Yaskawa INFORM job: X4_NOWY2_SPR.JBI

/JOB
//NAME X4_NOWY2_SPR
//POS
///NPOS 273,273,273,16,0,0
///TOOL 0
///POSTYPE PULSE
///PULSE
C00000=1579,-114561,-88072,141,60969,-160
C00001=1579,-126069,-115869,130,72161,-147
C00002=-67532,-124352,-115339,134,72718,-152
C00003=-81630,-76415,-67707,7081,99866,-75616
C00004=-81630,-76414,-67706,7081,99866,-75616
C00005=-84756,-88459,-71994,6618,96608,-76878
C00006=-84756,-88020,-70779,6612,96092,-76905
C00007=-84756,-88291,-71526,6619,96412,-76888
C00008=-86383,-83236,-69405,6430,97828,-77376
C00009=-86383,-82906,-68386,6422,97374,-77400
C00010=-85654,-85197,-69362,6508,96744,-77183
C00011=-88190,-77633,-68794,6246,100461,-77872
C00012=-91609,-64546,-67425,5952,106567,-78770
C00013=-108338,-72557,-69392,19017,102016,-84323
C00014=-103994,-87799,-70649,19047,94316,-83966
C00015=-101720,-95837,-73131,19200,91317,-83621
C00016=-101720,-95093,-71454,19192,90702,-83718
C00017=-101720,-95403,-72147,19196,90955,-83679
C00018=-102509,-90897,-70406,19144,92318,-83747
C00019=-102509,-90529,-69509,19136,91974,-83801
C00020=-102070,-93055,-70499,19166,91217,-83763
C00021=-103193,-87364,-70534,19135,94271,-83684
C00022=-105000,-74500,-64879,19101,97659,-83800
C00023=-113069,-60767,-53247,26239,106025,-84622
C00024=-112828,-63942,-52646,27281,108527,-83919
C00025=-112433,-69525,-54608,27546,108328,-83811
C00026=-112433,-69174,-53580,27467,107925,-83912
C00027=-112433,-68598,-51946,27347,107292,-84070
C00028=-112433,-68839,-52622,27396,107553,-84005
C00029=-112673,-65386,-50917,27452,108279,-83921
C00030=-112673,-65100,-50066,27387,107943,-84004
C00031=-112560,-66748,-50889,27360,107600,-84043
C00032=-112776,-63836,-50109,27476,108578,-83887
C00033=-126682,-57830,-51235,23795,116313,-87772
C00034=-91609,-64546,-67425,5952,106567,-78770
C00035=-73590,-134956,-134527,8565,110042,-72105
C00036=-73590,-134956,-134527,8565,110042,-72105
C00037=-85079,-90579,-82104,6699,101738,-76716
C00038=-105233,-99145,-78854,31145,91869,-85162
C00039=-90886,-100639,-75930,30232,80497,-82559
C00040=-84197,-95229,-69335,30102,76988,-80863
C00041=-84197,-94656,-68126,30150,76597,-80967
C00042=-84197,-94979,-68806,30123,76817,-80908
C00043=-86405,-88952,-66471,30068,79053,-81183
C00044=-86405,-88608,-65674,30094,78780,-81256
C00045=-85194,-91982,-67001,30129,77549,-81108
C00046=-89786,-90500,-68269,30172,80536,-82119
C00047=-91499,-86657,-71640,30020,84676,-81700
C00048=-78974,-84836,-79700,7511,102662,-74517
C00049=-78974,-83060,-72035,7396,98889,-74746
C00050=-78731,-83061,-70147,7399,97713,-74732
C00051=-78731,-82586,-68642,7386,97035,-74771
C00052=-78693,-82844,-69189,7365,97187,-74749
C00053=-80468,-78121,-67102,7173,98481,-75288
C00054=-80468,-77948,-66494,7167,98198,-75304
C00055=-79573,-80363,-67572,7265,97545,-75033
C00056=-80252,-78819,-67734,7202,98493,-75213
C00057=-80252,-80316,-73749,7282,101403,-75042
C00058=-98731,-93358,-79222,4709,99471,-81580
C00059=-97921,-96065,-76902,4782,96613,-81409
C00060=-97642,-96671,-75645,4808,95516,-81355
C00061=-97642,-96038,-74155,4803,94926,-81379
C00062=-97642,-96278,-74718,4805,95148,-81370
C00063=-99165,-88824,-71799,4613,97264,-81812
C00064=-99165,-88527,-70990,4608,96920,-81825
C00065=-98316,-92764,-72679,4715,95737,-81578
C00066=-99279,-88707,-72907,4606,98011,-81825
C00067=-99279,-90964,-80150,4662,101298,-81702
C00068=-83031,-73882,-65637,-17912,114082,-77307
C00069=-84799,-81323,-60919,-25592,110942,-77323
C00070=-87066,-81955,-59363,-24887,108536,-77734
C00071=-87066,-80978,-57100,-24746,107724,-77553
C00072=-87066,-81307,-57855,-24792,107993,-77613
C00073=-89010,-75270,-55192,-25677,108733,-78552
C00074=-89010,-74947,-54382,-25621,108431,-78482
C00075=-88073,-77930,-55720,-25197,108074,-78029
C00076=-86155,-69275,-53538,-25095,111477,-78039
C00077=-82305,-66217,-52035,-23871,113209,-76862
C00078=-98731,-93358,-79222,4709,99471,-81580
C00079=-87850,-130184,-128808,6122,98008,-77863
C00080=-131124,-97291,-82060,5244,66687,-6018
C00081=-125790,2337,-22266,13440,105024,83634
C00082=-119533,36956,22492,13071,94512,84678
C00083=-111606,23469,-6781,11265,89839,86812
C00084=-109349,27190,646,10801,86931,87307
C00085=-108816,27234,2830,10703,85564,87368
C00086=-108816,27153,4539,10716,84489,87276
C00087=-108816,27166,4149,10713,84731,87297
C00088=-107956,27551,4528,10540,84587,87578
C00089=-108965,27264,1619,10711,86335,87387
C00090=-111260,52324,24435,15027,98353,88139
C00091=-102462,56667,28820,9286,105586,72437
C00092=-101371,54153,30717,9255,103034,72626
C00093=-101300,53253,30624,9243,102627,72619
C00094=-101300,53374,32279,9201,101680,72548
C00095=-101300,53356,32072,9206,101797,72557
C00096=-100857,47625,25743,9281,102687,72780
C00097=-100773,46580,24617,9295,102831,72821
C00098=-101300,53356,32072,9206,101797,72557
C00099=-102175,52590,31226,9140,102021,72268
C00100=-102630,52208,30804,9106,102134,72116
C00101=-102175,52590,31226,9140,102021,72268
C00102=-99428,22928,-9812,4382,95874,-22555
C00103=-101546,17046,-6787,4678,91283,-23411
C00104=-101546,16945,-5416,4675,90390,-23444
C00105=-101514,16566,-4490,4670,89624,-23462
C00106=-101514,16574,-4727,4671,89774,-23457
C00107=-101796,19478,-2026,4708,89621,-23556
C00108=-101749,19095,-4432,4706,90897,-23492
C00109=-101749,19375,-7041,4715,92641,-23427
C00110=-101749,19375,-7041,4715,92641,-23427
C00111=-102981,33005,7118,6834,98538,-23358
C00112=-102660,29046,5283,6805,97611,-23301
C00113=-102660,29002,6609,6789,96777,-23347
C00114=-102660,29022,5897,6798,97224,-23322
C00115=-102541,27735,4980,6792,97060,-7882
C00116=-102724,29871,7085,6794,96879,-7954
C00117=-102669,29379,3677,6831,98706,-7835
C00118=-102669,30744,-3500,6979,103789,-7548
C00119=-89085,-61640,-68335,6227,95184,-3424
C00120=-129723,10180,-8133,7222,98462,-17027
C00121=-105913,33806,-16630,-33387,116609,-16888
C00122=-114766,23108,-3420,-30164,101829,-15972
C00123=-126000,19507,-6631,-29272,96237,-18805
C00124=-125928,21918,3078,-29245,93808,-18174
C00125=-125928,21960,4203,-29214,93219,-18024
C00126=-125927,21943,3808,-29209,93425,-18075
C00127=-125864,24512,6268,-29206,93280,-18014
C00128=-125884,23639,4506,-29235,93832,-18161
C00129=-125884,23787,-988,-29454,96866,-18937
C00130=-117200,23539,-1226,-29926,99884,-16393
C00131=-117161,21121,72,-29726,98116,-15912
C00132=-117144,20144,1246,-29621,97051,-15628
C00133=-117144,20183,2462,-29564,96414,-15463
C00134=-117144,20179,2362,-29568,96466,-15476
C00135=-117212,24135,6125,-29546,96194,-15431
C00136=-117202,23528,1396,-29761,98470,-16021
C00137=-113126,35471,9950,-29950,100652,-15017
C00138=-113126,35383,12410,-29782,99292,-14657
C00139=-113602,35282,14657,-29641,97872,-14469
C00140=-113602,35350,16056,-29571,97148,-14281
C00141=-113602,35312,15354,-29605,97509,-14375
C00142=-114294,35130,15170,-29602,97286,-14585
C00143=-113391,35371,15415,-29607,97577,-14310
C00144=-113626,42883,17073,-29878,99977,-15031
C00145=-136877,41374,10058,10283,103905,-75706
C00146=-141001,35831,8537,10150,102526,-77247
C00147=-140132,39057,14516,9459,103035,-76976
C00148=-140132,39037,16298,9412,101942,-77061
C00149=-140132,39036,16078,9417,102075,-77051
C00150=-140481,35058,11996,9419,102579,-77132
C00151=-140132,39036,16078,9417,102075,-77051
C00152=-138905,38111,15122,9481,102046,-76624
C00153=-140132,39045,14975,9447,102749,-76998
C00154=-140132,39114,13214,9498,103853,-76912
C00155=-141320,33353,7524,13959,97601,-77374
C00156=-139853,30861,8005,10213,95427,-68773
C00157=-139850,30231,7379,10216,95489,-68766
C00158=-141726,26843,4526,13791,96694,-77632
C00159=-141207,31872,9522,12754,100191,-77170
C00160=-131838,40307,17400,-3069,104254,-75449
C00161=-120717,39791,20254,-22002,103322,-74072
C00162=-123241,41817,22993,-23858,102713,-75145
C00163=-120965,41759,25023,-29185,101758,-74907
C00164=-121023,25271,5223,-28433,95326,-73297
C00165=-120372,33506,8504,-28624,97501,-73589
C00166=-120372,33506,8504,-28624,97501,-7388
C00167=-114011,28987,3831,-29482,105348,-6966
C00168=-127301,22883,-362,-9290,98378,-8800
C00169=-130383,22892,110,-12210,96784,-9925
C00170=-119117,21486,5591,-32037,93907,-6966
C00171=-117872,21036,1539,-32238,96305,-7157
C00172=-135561,25772,-1454,-7801,99682,-11540
C00173=-135461,26025,2407,-7746,97466,-11367
C00174=-129197,23357,2778,-20865,94605,-10044
C00175=-129563,23522,5318,-26932,92135,-10188
C00176=-126533,22338,1333,-27220,94758,-9659
C00177=-115633,44815,18495,-18996,108364,22675
C00178=-114062,50158,32326,-24769,103985,23625
C00179=-114261,61004,44440,-24574,102207,23931
C00180=-113327,59043,39697,-24681,104230,23854
C00181=-113549,43239,22387,-25049,106471,23276
C00182=-113959,36250,17368,-26116,100180,17331
C00183=-113750,32141,13338,-26671,97959,14884
C00184=-113784,32033,10394,-26825,99526,14508
C00185=-112924,58292,37776,-24734,105077,23825
C00186=-109456,25709,2980,-23794,97137,26657
C00187=-118237,30699,-4511,6400,110959,24971
C00188=-106534,-87247,-110627,560,89262,27492
C00189=-106534,-87247,-110627,560,89262,27492
C00190=-103790,-60662,-71601,3492,92371,24893
C00191=-90072,-46297,-51679,19403,82444,29914
C00192=-89225,-25796,-38496,19051,95364,28629
C00193=-82968,-19569,-33829,18693,94249,30668
C00194=-92316,-28208,-34631,31848,87681,26801
C00195=-93212,-29211,-40642,31971,90742,27310
C00196=-74629,-7827,-31935,11254,101997,33705
C00197=-71338,-2997,-23236,6798,101883,34323
C00198=-78936,-14568,-30649,16904,94877,32031
C00199=-82428,-18766,-28557,29607,85533,29992
C00200=-85091,-23046,-35219,29948,88128,29642
C00201=-83302,-13788,-26964,29706,87219,30090
C00202=-84406,-14503,-30600,29861,89239,30192
C00203=-85356,-5858,-28119,20956,91780,-33865
C00204=-81588,1907,-17110,16920,91332,-34481
C00205=-80085,-4136,-22119,16745,91007,-34003
C00206=-79500,-6857,-23987,16670,90650,-33848
C00207=-76840,-15565,-30031,18766,92661,-32418
C00208=-81974,-12051,-30981,19262,96095,-33689
C00209=-98247,-31422,-44950,19682,96659,-36405
C00210=-99612,-12458,-27594,19698,96098,-36983
C00211=-98475,-20893,-33899,19626,95400,-36692
C00212=-97436,-32531,-42916,18662,91677,-32211
C00213=-95696,-34091,-42802,18103,89563,-30497
C00214=-96230,-30895,-40673,18159,89998,-30622
C00215=-92776,-41331,-47434,14269,83214,-21666
C00216=-93749,-43799,-52657,14401,85273,-21763
C00217=-91043,-39779,-53377,13904,87247,-20611
C00218=-86158,-7385,-30463,15366,102993,-69398
C00219=-78323,6041,-20316,6463,111515,-89101
C00220=-75958,-7074,-26718,1279,101463,-89171
C00221=-73720,-14383,-32408,1291,101175,-88413
C00222=-73707,-14423,-32438,1291,101173,-88409
C00223=-74501,-16417,-33720,1350,100398,-77182
C00224=-81364,-12014,-29075,8477,103574,-60369
C00225=-76974,-6126,-24441,8683,103288,-58863
C00226=-85840,-5383,-30241,8443,108111,-61612
C00227=-85618,-23129,-54211,-23,98050,-63088
C00228=-77730,-75302,-67065,7588,99691,-74263
C00229=-69151,-69068,-61329,2748,102842,-72431
C00230=-87447,-85862,-67970,-5918,101111,-78781
C00231=-86539,-83533,-63306,-15976,104237,-78477
C00232=-79657,-74315,-62077,-14413,109372,-76594
C00233=-66263,-128090,-130023,-6185,104579,-72041
C00234=-66263,-128090,-130023,-6185,104579,-72041
C00235=-94568,-90015,-76427,-6942,102962,-81955
C00236=-117602,-94880,-71794,-18297,96358,-89322
C00237=-121559,-93963,-69420,-18891,94518,-90455
C00238=-120999,-73428,-51402,-33795,103006,-79102
C00239=-123309,-67068,-41693,-44286,101999,-75160
C00240=-127601,-64996,-39493,-46701,100367,-75399
C00241=-114717,-64735,-41398,-43474,107786,-72608
C00242=-113328,-78138,-63059,-20614,107376,-72751
C00243=-119967,-79989,-67356,5538,106972,-75179
C00244=-119600,-81312,-64641,5556,104608,-75155
C00245=-101370,-77587,-62989,10017,103725,-68716
C00246=-107781,-79603,-61547,20378,100372,-71634
C00247=-114949,-81063,-65452,19014,103658,-73736
C00248=-107597,-133050,-132520,1199,109480,-70827
C00249=-107600,-133050,-132519,1199,109480,-70827
C00250=-111097,-94755,-74427,15472,95771,-72593
C00251=-108511,-92825,-70401,15771,93843,-71925
C00252=-108472,-92930,-69979,15769,93534,-71951
C00253=-101455,-63185,-52092,14913,110854,-65885
C00254=-99527,-62495,-51665,15536,110582,-65187
C00255=-84477,-52236,-46062,20087,109018,-59662
C00256=-81486,-46306,-41350,23406,108929,-56767
C00257=-85967,-47236,-42901,22323,110616,-58192
C00258=-110623,-74300,-66049,9174,91324,-69507
C00259=-118006,-113386,-124466,9637,107827,-70792
C00260=-118006,-113386,-124466,9637,107827,-70792
C00261=-104411,-100441,-71960,6543,87095,-88178
C00262=-104969,-99438,-67477,6508,84909,-88479
C00263=-110340,-97663,-63190,-18251,87254,-88347
C00264=-100177,-101375,-72775,-10447,90542,-85701
C00265=-127322,-146784,-131564,384,102103,-77635
C00266=-127322,-146784,-131564,384,102103,-77635
C00267=-128828,-100845,-70585,1227,88109,-75124
C00268=-127499,-98820,-66694,1376,86733,-74692
C00269=-112766,-97884,-65315,11280,85320,-70490
C00270=-128822,-103835,-77575,9498,91788,-75427
C00271=-146076,-192209,-136001,7129,84184,-81740
C00272=-146076,-192209,-136001,7129,84184,-81740
BC00000=127053,672594,1075229
BC00001=127053,672594,1075229
BC00002=210750,818892,1075229
BC00003=210750,818892,1005167
BC00004=210749,818892,1005164
BC00005=210749,818892,1005161
BC00006=210749,818892,1005161
BC00007=210749,818892,1005161
BC00008=210749,818892,1005161
BC00009=210749,818892,1005161
BC00010=210749,818892,1005161
BC00011=210749,818892,1005161
BC00012=210749,818892,1005161
BC00013=255741,818892,1005161
BC00014=255741,818892,1005161
BC00015=255741,818892,1005161
BC00016=255741,818892,1005161
BC00017=255741,818892,1005161
BC00018=255741,818892,1005161
BC00019=255741,818892,1005161
BC00020=255741,818892,1005161
BC00021=255741,818892,1005161
BC00022=255741,818892,1005161
BC00023=287623,818892,1005161
BC00024=287623,818892,1005161
BC00025=287623,818892,1005161
BC00026=287623,818892,1005161
BC00027=287623,818892,1005161
BC00028=287623,818892,1005161
BC00029=287623,818892,1005161
BC00030=287623,818892,1005161
BC00031=287623,818892,1005161
BC00032=287623,818892,1005161
BC00033=287623,818892,1005161
BC00034=210749,818892,1005161
BC00035=210749,818892,1005161
BC00036=119260,818892,1005161
BC00037=119260,818892,1005161
BC00038=119260,818892,1005161
BC00039=119260,818892,1005161
BC00040=119260,818892,1005161
BC00041=119260,818892,1005161
BC00042=119260,818892,1005161
BC00043=119260,818892,1005161
BC00044=119260,818892,1005161
BC00045=119260,818892,1005161
BC00046=119260,818892,1005161
BC00047=119260,818892,1005161
BC00048=119260,818892,1005157
BC00049=119260,818892,1005157
BC00050=119260,818892,1005157
BC00051=119260,818892,1005157
BC00052=119260,818892,1005157
BC00053=119260,818892,1005157
BC00054=119260,818892,1005157
BC00055=119260,818892,1005157
BC00056=119260,818892,1005157
BC00057=119260,818892,1005157
BC00058=119260,818892,1005157
BC00059=119260,818892,1005157
BC00060=119260,818892,1005157
BC00061=119260,818892,1005157
BC00062=119260,818892,1005157
BC00063=119260,818892,1005157
BC00064=119260,818892,1005157
BC00065=119260,818892,1005157
BC00066=119260,818892,1005157
BC00067=119260,818892,1005157
BC00068=119260,818892,1005157
BC00069=119260,818892,1005157
BC00070=119260,818892,1005157
BC00071=119260,818892,1005157
BC00072=119260,818892,1005157
BC00073=119260,818892,1005157
BC00074=119260,818892,1005157
BC00075=119260,818892,1005157
BC00076=119260,818892,1005157
BC00077=119260,818892,1005157
BC00078=119260,818892,1005157
BC00079=119260,818892,1005157
BC00080=271066,672595,967916
BC00081=271066,672595,967916
BC00082=271066,672595,967916
BC00083=271066,672595,742596
BC00084=271066,672596,742593
BC00085=271066,672596,742593
BC00086=271065,672596,742589
BC00087=271065,672596,742589
BC00088=271065,672596,742589
BC00089=271065,672597,742586
BC00090=271065,672597,742586
BC00091=271065,673087,742586
BC00092=271065,673087,742586
BC00093=271065,673087,742586
BC00094=271065,673087,742586
BC00095=271065,673087,742586
BC00096=271065,673087,742586
BC00097=271065,673087,742586
BC00098=271065,673087,742586
BC00099=271065,673087,742586
BC00100=271065,673087,742586
BC00101=271065,673087,742586
BC00102=271065,673085,742583
BC00103=271065,673085,742583
BC00104=271065,673085,742583
BC00105=271065,673085,742583
BC00106=271065,673085,742583
BC00107=271065,673085,742583
BC00108=271065,673085,742583
BC00109=271065,673085,742583
BC00110=291623,673085,742583
BC00111=291623,673085,742583
BC00112=291623,673085,742583
BC00113=291623,673085,742583
BC00114=291623,673085,742583
BC00115=291623,673085,742583
BC00116=291623,673085,742583
BC00117=291623,673085,742583
BC00118=291623,673085,1054355
BC00119=130801,673085,1059449
BC00120=130802,673083,1031676
BC00121=130802,673083,742569
BC00122=130802,673083,742569
BC00123=130802,673083,742569
BC00124=130802,673083,742569
BC00125=130802,673083,742569
BC00126=130802,673083,742566
BC00127=130802,673083,742566
BC00128=130802,673083,742566
BC00129=130802,673083,742566
BC00130=130802,673083,742566
BC00131=130802,673083,742566
BC00132=130802,673083,742566
BC00133=130802,673083,742566
BC00134=130802,673083,742566
BC00135=130802,673083,742566
BC00136=130802,673083,742566
BC00137=130802,673083,742566
BC00138=130802,673083,742566
BC00139=130802,673083,742566
BC00140=130802,673083,742566
BC00141=130802,673083,742566
BC00142=130802,673083,742566
BC00143=130802,673083,742566
BC00144=130802,673083,742566
BC00145=130802,673083,742566
BC00146=130802,673083,742566
BC00147=130802,673083,742566
BC00148=130802,673083,742566
BC00149=130802,673083,742566
BC00150=130802,673083,742566
BC00151=130802,673083,742566
BC00152=130802,673083,742566
BC00153=130802,673083,742566
BC00154=130802,673083,742566
BC00155=130802,673083,742566
BC00156=130802,673083,742566
BC00157=130802,673083,742566
BC00158=130802,673083,742566
BC00159=130802,673083,742566
BC00160=130802,673083,742566
BC00161=130802,673083,742566
BC00162=130802,673083,742566
BC00163=130802,673083,742566
BC00164=130802,673083,742566
BC00165=130802,673083,742566
BC00166=130802,673083,742566
BC00167=130802,673083,742566
BC00168=130802,673083,742566
BC00169=130802,673083,742566
BC00170=130802,673083,742566
BC00171=130802,673083,742566
BC00172=130802,673083,742566
BC00173=130802,673083,742566
BC00174=130802,673083,742566
BC00175=130802,673083,742566
BC00176=130802,673083,742566
BC00177=130802,673083,742566
BC00178=130802,673083,742566
BC00179=130802,673083,742566
BC00180=130802,673083,742566
BC00181=130802,673083,742566
BC00182=130802,673083,742566
BC00183=130802,673083,742566
BC00184=130802,673083,742566
BC00185=130802,673083,742566
BC00186=130802,673083,742566
BC00187=130802,673083,742566
BC00188=130802,673083,742566
BC00189=239197,673083,742566
BC00190=239197,748715,742566
BC00191=239197,748715,742566
BC00192=239196,748714,742562
BC00193=239196,748714,742562
BC00194=239196,748714,742562
BC00195=239196,748714,742562
BC00196=239196,748714,742562
BC00197=239196,748714,742562
BC00198=239196,748714,742562
BC00199=239196,748714,742562
BC00200=239196,748714,742562
BC00201=239196,748714,742562
BC00202=239196,748714,742559
BC00203=239196,748714,742559
BC00204=239196,748714,742559
BC00205=239196,748714,742559
BC00206=239196,748714,742559
BC00207=239196,748714,742559
BC00208=239196,748714,742559
BC00209=239196,748714,742559
BC00210=239196,748714,742559
BC00211=239196,748714,742559
BC00212=239196,748714,742559
BC00213=239196,748714,742559
BC00214=239196,748714,742559
BC00215=239196,748714,742559
BC00216=239196,748714,742559
BC00217=239196,748714,742559
BC00218=239196,748714,742559
BC00219=239196,748714,742559
BC00220=239196,748714,742559
BC00221=239196,748714,742559
BC00222=239196,748714,742559
BC00223=239196,748714,742559
BC00224=239196,748714,742559
BC00225=239196,748714,742559
BC00226=239196,748714,742559
BC00227=239196,748714,742556
BC00228=210749,818892,1005161
BC00229=210749,818892,1005161
BC00230=210750,818891,1005159
BC00231=210750,818891,1005159
BC00232=210750,818891,1005159
BC00233=210750,818891,1005157
BC00234=123072,818891,1005157
BC00235=123072,818891,1005157
BC00236=162220,818891,1005157
BC00237=162220,818891,1005152
BC00238=162220,818891,1005153
BC00239=162220,818891,1005153
BC00240=162220,818891,1005153
BC00241=162220,818891,1005153
BC00242=162220,818891,1005153
BC00243=162220,818891,1005153
BC00244=162220,818891,1005153
BC00245=162220,818891,1005153
BC00246=162220,818891,1005153
BC00247=162220,818891,1005153
BC00248=162220,818891,1005153
BC00249=264269,818892,1005150
BC00250=264269,818892,1005150
BC00251=264269,818892,1005150
BC00252=264269,818892,1005148
BC00253=264269,818892,1005148
BC00254=264269,818892,1005148
BC00255=264269,818892,1005148
BC00256=264269,818892,1005148
BC00257=264269,818892,1005148
BC00258=264269,818892,1005148
BC00259=264269,818892,1005148
BC00260=150431,818892,1056877
BC00261=150431,818892,1056877
BC00262=150431,818892,1056877
BC00263=150431,818892,1056877
BC00264=150431,818892,1056877
BC00265=150431,818892,1056877
BC00266=276083,818892,1056877
BC00267=276083,818892,1056877
BC00268=276083,818892,1056877
BC00269=276083,818892,1056877
BC00270=276083,818892,1056877
BC00271=276083,818892,1056877
BC00272=276083,684480,1056877
EC00000=-1527674,557300
EC00001=-1527674,557300
EC00002=-1527674,557300
EC00003=-1527674,557300
EC00004=-1527674,557300
EC00005=-1527674,557301
EC00006=-1527674,557301
EC00007=-1527674,557301
EC00008=-1527674,557301
EC00009=-1527674,557301
EC00010=-1527674,557301
EC00011=-1527674,557301
EC00012=-1527674,557301
EC00013=-1527674,557301
EC00014=-1527674,557301
EC00015=-1527674,557301
EC00016=-1527674,557301
EC00017=-1527674,557301
EC00018=-1527674,557301
EC00019=-1527674,557301
EC00020=-1527674,557301
EC00021=-1527674,557301
EC00022=-1527674,557301
EC00023=-1527674,557301
EC00024=-1527674,557301
EC00025=-1527674,557301
EC00026=-1527674,557301
EC00027=-1527674,557301
EC00028=-1527674,557301
EC00029=-1527674,557301
EC00030=-1527674,557301
EC00031=-1527674,557301
EC00032=-1527674,557301
EC00033=-1527674,557301
EC00034=-1527674,557301
EC00035=-1527674,557301
EC00036=-1527674,557301
EC00037=-1527674,557301
EC00038=-1527674,557301
EC00039=-1527674,557301
EC00040=-1527674,557301
EC00041=-1527674,557301
EC00042=-1527674,557301
EC00043=-1527674,557301
EC00044=-1527674,557301
EC00045=-1527674,557301
EC00046=-1527674,557301
EC00047=-1527674,557301
EC00048=-1527675,557301
EC00049=-1527675,557301
EC00050=-1527675,557301
EC00051=-1527675,557301
EC00052=-1527675,557301
EC00053=-1527675,557301
EC00054=-1527675,557301
EC00055=-1527675,557301
EC00056=-1527675,557301
EC00057=-1527675,557301
EC00058=-1527675,557301
EC00059=-1527675,557301
EC00060=-1527675,557301
EC00061=-1527675,557301
EC00062=-1527675,557301
EC00063=-1527675,557301
EC00064=-1527675,557301
EC00065=-1527675,557301
EC00066=-1527675,557301
EC00067=-1527675,557301
EC00068=-1527675,557301
EC00069=-1527675,557301
EC00070=-1527675,557301
EC00071=-1527675,557301
EC00072=-1527675,557301
EC00073=-1527675,557301
EC00074=-1527675,557301
EC00075=-1527675,557301
EC00076=-1527675,557301
EC00077=-1527675,557301
EC00078=-1527675,557301
EC00079=-1527675,557301
EC00080=-1332361,557301
EC00081=-1332361,557301
EC00082=-1332361,557301
EC00083=-1332361,557301
EC00084=-1332361,557302
EC00085=-1332361,557302
EC00086=-1332361,557302
EC00087=-1332361,557302
EC00088=-1332361,557302
EC00089=-1332361,557302
EC00090=-1332361,557302
EC00091=-1332361,557302
EC00092=-1332361,557302
EC00093=-1332361,557302
EC00094=-1332361,557302
EC00095=-1332361,557302
EC00096=-1332361,557302
EC00097=-1332361,557302
EC00098=-1332361,557302
EC00099=-1332361,557302
EC00100=-1332361,557302
EC00101=-1332361,557302
EC00102=-1332361,557302
EC00103=-1332361,557302
EC00104=-1332361,557302
EC00105=-1332361,557302
EC00106=-1332361,557302
EC00107=-1332361,557302
EC00108=-1332361,557302
EC00109=-1332361,557302
EC00110=-1332361,557302
EC00111=-1332361,557302
EC00112=-1332361,557302
EC00113=-1332361,557302
EC00114=-1332361,557302
EC00115=-1332361,557302
EC00116=-1332361,557302
EC00117=-1332361,557302
EC00118=-1332361,557302
EC00119=-1332361,557302
EC00120=-1332361,557303
EC00121=-1332361,557303
EC00122=-1332361,557303
EC00123=-1332361,557303
EC00124=-1332361,557303
EC00125=-1332361,557303
EC00126=-1332361,557303
EC00127=-1332361,557303
EC00128=-1332361,557303
EC00129=-1332361,557303
EC00130=-1332361,557303
EC00131=-1332361,557303
EC00132=-1332361,557303
EC00133=-1332361,557303
EC00134=-1332361,557303
EC00135=-1332361,557303
EC00136=-1332361,557303
EC00137=-1332361,557303
EC00138=-1332361,557303
EC00139=-1332361,557303
EC00140=-1332361,557303
EC00141=-1332361,557303
EC00142=-1332361,557303
EC00143=-1332361,557303
EC00144=-1332361,557303
EC00145=-1332361,557303
EC00146=-1332361,557303
EC00147=-1332361,557303
EC00148=-1332361,557303
EC00149=-1332361,557303
EC00150=-1332361,557303
EC00151=-1332361,557303
EC00152=-1332361,557303
EC00153=-1332361,557303
EC00154=-1332361,557303
EC00155=-1332361,557303
EC00156=-1332361,557303
EC00157=-1332361,557303
EC00158=-1332361,557303
EC00159=-1332361,557303
EC00160=-1332361,557303
EC00161=-1332361,557303
EC00162=-1332361,557303
EC00163=-1332361,557303
EC00164=-1332361,557303
EC00165=-1332361,557303
EC00166=-1332361,557303
EC00167=-1332361,557303
EC00168=-1332361,557303
EC00169=-1332361,557303
EC00170=-1332361,557303
EC00171=-1332361,557303
EC00172=-1332361,557303
EC00173=-1332361,557303
EC00174=-1332361,557303
EC00175=-1332361,557303
EC00176=-1332361,557303
EC00177=-1332361,557303
EC00178=-1332361,557303
EC00179=-1332361,557303
EC00180=-1332361,557303
EC00181=-1332361,557303
EC00182=-1332361,557303
EC00183=-1332361,557303
EC00184=-1332361,557303
EC00185=-1332361,557303
EC00186=-1332361,557303
EC00187=-1332361,557303
EC00188=-1332361,557303
EC00189=-1332361,557303
EC00190=-1332361,557303
EC00191=-1332361,557303
EC00192=-1332361,557303
EC00193=-1332361,557303
EC00194=-1332361,557303
EC00195=-1332361,557303
EC00196=-1332361,557303
EC00197=-1332361,557303
EC00198=-1332361,557303
EC00199=-1332361,557303
EC00200=-1332361,557303
EC00201=-1332361,557303
EC00202=-1332361,557303
EC00203=-1332361,557303
EC00204=-1332361,557303
EC00205=-1332361,557303
EC00206=-1332361,557303
EC00207=-1332361,557303
EC00208=-1332361,557303
EC00209=-1332361,557303
EC00210=-1332361,557303
EC00211=-1332361,557303
EC00212=-1332361,557303
EC00213=-1332361,557303
EC00214=-1332361,557303
EC00215=-1332361,557303
EC00216=-1332361,557303
EC00217=-1332361,557303
EC00218=-1332361,557303
EC00219=-1332361,557303
EC00220=-1332361,557303
EC00221=-1332361,557303
EC00222=-1332361,557303
EC00223=-1332361,557303
EC00224=-1332361,557303
EC00225=-1332361,557303
EC00226=-1332361,557303
EC00227=-1332361,557303
EC00228=-1527674,557301
EC00229=-1527674,557301
EC00230=-1527675,557301
EC00231=-1527675,557301
EC00232=-1527675,557301
EC00233=-1527675,557302
EC00234=-1527675,557302
EC00235=-1527675,557302
EC00236=-1527675,557302
EC00237=-1527676,557302
EC00238=-1527676,557302
EC00239=-1527676,557302
EC00240=-1527676,557302
EC00241=-1527676,557302
EC00242=-1527676,557302
EC00243=-1527676,557302
EC00244=-1527676,557302
EC00245=-1527676,557302
EC00246=-1527676,557302
EC00247=-1527676,557302
EC00248=-1527676,557302
EC00249=-1527677,557302
EC00250=-1527677,557302
EC00251=-1527677,557302
EC00252=-1527678,557302
EC00253=-1527678,557302
EC00254=-1527678,557302
EC00255=-1527678,557302
EC00256=-1527678,557302
EC00257=-1527678,557302
EC00258=-1527678,557302
EC00259=-1527678,557302
EC00260=-1527678,557302
EC00261=-1527678,557302
EC00262=-1527678,557302
EC00263=-1527678,557302
EC00264=-1527678,557302
EC00265=-1527678,557302
EC00266=-1527678,557302
EC00267=-1527678,557302
EC00268=-1527678,557302
EC00269=-1527678,557302
EC00270=-1527678,557302
EC00271=-1527678,557302
EC00272=-1527678,557302
///POSTYPE BASE
///RECTAN
///RCONF 0,0,0,0,0,0,0,0,0,0,0,0,0,0,0,0,0,0,0,0,0,0,0,0
P00006=0.222,-3.123,-1.508,0.0000,0.0000,0.0000
P00021=-0.225,-6.128,-0.405,0.0000,0.0000,0.0000
P00022=0.222,-3.123,-1.508,0.0000,0.0000,0.0000
P00023=0.143,-0.036,0.682,0.0000,0.0000,0.0000
P00024=0.145,-0.552,1.326,0.0000,0.0000,0.0000
P00025=-2.003,0.006,0.728,0.0000,0.0000,0.0000
P00026=0.562,-0.002,-0.337,0.0000,0.0000,0.0000
P00027=-0.746,0.015,-9.096,0.0000,0.0000,0.0000
P00031=1.853,-0.001,-1.549,0.0000,0.0000,0.0000
P00032=1.957,0.503,-7.217,0.0000,0.0000,0.0000
///RCONF 0,0,0,0,1,0,0,0,0,0,0,0,0,0,0,0,0,0,0,0,0,0,0,0
P00033=-0.123,0.612,-5.012,0.0000,0.0000,0.0000
///RCONF 0,0,0,0,0,0,0,0,0,0,0,0,0,0,0,0,0,0,0,0,0,0,0,0
P00034=-0.304,0.773,-2.693,0.0000,0.0000,0.0000
P00035=2.817,0.591,-1.622,0.0000,0.0000,0.0000
P00036=-1.108,-0.829,1.850,0.0000,0.0000,0.0000
P00037=0.023,0.937,-2.677,0.0000,0.0000,0.0000
P00038=0.158,-1.133,-1.952,0.0000,0.0000,0.0000
//INST
///DATE 2024/04/03 18:26
///ATTR SC,RW
///GROUP1 RB1,BS1
///GROUP2 ST1
NOP
'PIERWSZA SEKWENCJA
MOVJ C00000 BC00000 VJ=100.00  +MOVJ EC00000 VJ=100.00
MOVJ C00001 BC00001 VJ=100.00  +MOVJ EC00001 VJ=100.00
MOVJ C00002 BC00002 VJ=100.00  +MOVJ EC00002 VJ=100.00
MOVJ C00003 BC00003 VJ=100.00  +MOVJ EC00003 VJ=100.00
SMOVL C00004 BC00004 V=166.7  +MOVJ EC00004
SMOVL C00005 BC00005 V=100.0  +MOVJ EC00005
SREFP 3 C00006 BC00006  +REFP EC00006
CALL JOB:SEARCH-R1-S13D
SET P021 P006
SFTON3D P021
SMOVL C00007 BC00007 V=100.0  +MOVJ EC00007
SMOVL C00008 BC00008 V=100.0  +MOVJ EC00008
SMOVL C00009 BC00009 V=100.0  +MOVJ EC00009
SREFP 3 C00010 BC00010  +REFP EC00010
CALL JOB:SEARCH-R1-S13D
SET P021 P006
SFTON3D P021
SMOVL C00011 BC00011 V=100.0  +MOVJ EC00011
MOVL C00012 BC00012 V=400.0  +MOVJ EC00012 VJ=100.00
SFTOF3D
SMOVL C00013 BC00013 V=1000.0  +MOVJ EC00013
SMOVL C00014 BC00014 V=166.7  +MOVJ EC00014
SMOVL C00015 BC00015 V=100.0  +MOVJ EC00015
SREFP 3 C00016 BC00016  +REFP EC00016
CALL JOB:SEARCH-R1-S13D
SET P022 P006
SFTON3D P022
SMOVL C00017 BC00017 V=100.0  +MOVJ EC00017
SMOVL C00018 BC00018 V=100.0  +MOVJ EC00018
SMOVL C00019 BC00019 V=100.0  +MOVJ EC00019
SREFP 3 C00020 BC00020  +REFP EC00020
CALL JOB:SEARCH-R1-S13D
SET P022 P006
SFTON3D P022
SMOVL C00021 BC00021 V=100.0  +MOVJ EC00021
MOVL C00022 BC00022 V=400.0  +MOVJ EC00022 VJ=100.00
SFTOF3D
SMOVL C00023 BC00023 V=1000.0  +MOVJ EC00023
SMOVL C00024 BC00024 V=400.0  +MOVJ EC00024
SMOVL C00025 BC00025 V=166.7  +MOVJ EC00025
SMOVL C00026 BC00026 V=100.0  +MOVJ EC00026
SREFP 3 C00027 BC00027  +REFP EC00027
CALL JOB:SEARCH-R1-S13D
SET P023 P006
SFTON3D P023
SMOVL C00028 BC00028 V=100.0  +MOVJ EC00028
SMOVL C00029 BC00029 V=100.0  +MOVJ EC00029
SMOVL C00030 BC00030 V=100.0  +MOVJ EC00030
SREFP 3 C00031 BC00031  +REFP EC00031
CALL JOB:SEARCH-R1-S13D
SET P023 P006
SFTON3D P023
SMOVL C00032 BC00032 V=100.0  +MOVJ EC00032
MOVL C00033 BC00033 V=400.0  +MOVJ EC00033 VJ=100.00
SFTOF3D
SMOVL C00034 BC00034 V=400.0  +MOVJ EC00034
MOVJ C00035 BC00035 VJ=100.00  +MOVJ EC00035 VJ=100.00
SMOVL C00036 BC00036 V=1000.0  +MOVJ EC00036
SMOVL C00037 BC00037 V=1000.0  +MOVJ EC00037
SMOVL C00038 BC00038 V=1000.0  +MOVJ EC00038
SMOVL C00039 BC00039 V=166.7  +MOVJ EC00039
SMOVL C00040 BC00040 V=100.0  +MOVJ EC00040
SREFP 3 C00041 BC00041  +REFP EC00041
CALL JOB:SEARCH-R1-S13D
SET P024 P006
SFTON3D P024
SMOVL C00042 BC00042 V=100.0  +MOVJ EC00042
SMOVL C00043 BC00043 V=100.0  +MOVJ EC00043
SMOVL C00044 BC00044 V=100.0  +MOVJ EC00044
SREFP 3 C00045 BC00045  +REFP EC00045
CALL JOB:SEARCH-R1-S13D
SET P024 P006
SFTON3D P024
SMOVL C00046 BC00046 V=100.0  +MOVJ EC00046
MOVL C00047 BC00047 V=400.0  +MOVJ EC00047 VJ=100.00
SMOVL C00048 BC00048 V=1000.0  +MOVJ EC00048
SMOVL C00049 BC00049 V=166.7  +MOVJ EC00049
SMOVL C00050 BC00050 V=100.0  +MOVJ EC00050
SREFP 3 C00051 BC00051  +REFP EC00051
CALL JOB:SEARCH-R1-S13D
SET P025 P006
SFTON3D P025
SMOVL C00052 BC00052 V=100.0  +MOVJ EC00052
SMOVL C00053 BC00053 V=100.0  +MOVJ EC00053
SMOVL C00054 BC00054 V=100.0  +MOVJ EC00054
SREFP 3 C00055 BC00055  +REFP EC00055
CALL JOB:SEARCH-R1-S13D
SET P025 P006
SFTON3D P025
SMOVL C00056 BC00056 V=100.0  +MOVJ EC00056
MOVL C00057 BC00057 V=400.0  +MOVJ EC00057 VJ=100.00
SFTOF3D
SMOVL C00058 BC00058 V=1000.0  +MOVJ EC00058
SMOVL C00059 BC00059 V=166.7  +MOVJ EC00059
SMOVL C00060 BC00060 V=100.0  +MOVJ EC00060
SREFP 3 C00061 BC00061  +REFP EC00061
CALL JOB:SEARCH-R1-S13D
SET P026 P006
SFTON3D P026
SMOVL C00062 BC00062 V=100.0  +MOVJ EC00062
SMOVL C00063 BC00063 V=100.0  +MOVJ EC00063
SMOVL C00064 BC00064 V=100.0  +MOVJ EC00064
SREFP 3 C00065 BC00065  +REFP EC00065
CALL JOB:SEARCH-R1-S13D
SET P026 P006
SFTON3D P026
SMOVL C00066 BC00066 V=100.0  +MOVJ EC00066
MOVL C00067 BC00067 V=400.0  +MOVJ EC00067 VJ=100.00
SFTOF3D
SMOVL C00068 BC00068 V=1000.0  +MOVJ EC00068
SMOVL C00069 BC00069 V=166.7  +MOVJ EC00069
SMOVL C00070 BC00070 V=100.0  +MOVJ EC00070
SREFP 3 C00071 BC00071  +REFP EC00071
CALL JOB:SEARCH-R1-S13D
SET P027 P006
SFTON3D P027
SMOVL C00072 BC00072 V=100.0  +MOVJ EC00072
SMOVL C00073 BC00073 V=100.0  +MOVJ EC00073
SMOVL C00074 BC00074 V=100.0  +MOVJ EC00074
SREFP 3 C00075 BC00075  +REFP EC00075
CALL JOB:SEARCH-R1-S13D
SET P027 P006
SFTON3D P027
SMOVL C00076 BC00076 V=100.0  +MOVJ EC00076
MOVL C00077 BC00077 V=400.0  +MOVJ EC00077 VJ=100.00
SFTOF3D
SMOVL C00078 BC00078 V=1000.0  +MOVJ EC00078
MOVJ C00079 BC00079 VJ=80.00  +MOVJ EC00079 VJ=80.00
'DRUGA SEKWENCJA
MOVJ C00080 BC00080 VJ=100.00  +MOVJ EC00080 VJ=100.00
MOVJ C00081 BC00081 VJ=100.00  +MOVJ EC00081 VJ=100.00
MOVJ C00082 BC00082 VJ=100.00  +MOVJ EC00082 VJ=100.00
SMOVL C00083 BC00083 V=1000.0  +MOVJ EC00083
SMOVL C00084 BC00084 V=166.7  +MOVJ EC00084
SMOVL C00085 BC00085 V=100.0  +MOVJ EC00085
SREFP 3 C00086 BC00086  +REFP EC00086
CALL JOB:SEARCH-R1-S13D
SET P031 P006
SFTON3D P031
SMOVL C00087 BC00087 V=100.0  +MOVJ EC00087
SREFP 3 C00088 BC00088  +REFP EC00088
CALL JOB:SEARCH-R1-S13D
SET P031 P006
SFTON3D P031
SMOVL C00089 BC00089 V=100.0  +MOVJ EC00089
MOVL C00090 BC00090 V=400.0  +MOVJ EC00090 VJ=100.00
SMOVL C00091 BC00091 V=1000.0  +MOVJ EC00091
SFTOF3D
SMOVL C00092 BC00092 V=166.7  +MOVJ EC00092
SMOVL C00093 BC00093 V=100.0  +MOVJ EC00093
SREFP 3 C00094 BC00094  +REFP EC00094
CALL JOB:SEARCH-R1-S13D
SET P032 P006
SFTON3D P032
SMOVL C00095 BC00095 V=100.0  +MOVJ EC00095
SMOVL C00096 BC00096 V=100.0  +MOVJ EC00096
SREFP 3 C00097 BC00097  +REFP EC00097
CALL JOB:SEARCH-R1-S13D
SET P032 P006
SFTON3D P032
SMOVL C00098 BC00098 V=100.0  +MOVJ EC00098
SMOVL C00099 BC00099 V=100.0  +MOVJ EC00099
SREFP 3 C00100 BC00100  +REFP EC00100
CALL JOB:SEARCH-R1-S13D
SET P032 P006
SFTON3D P032
SMOVL C00101 BC00101 V=100.0  +MOVJ EC00101
MOVL C00102 BC00102 V=400.0  +MOVJ EC00102 VJ=100.00
SFTOF3D
SMOVL C00103 BC00103 V=166.7  +MOVJ EC00103
SMOVL C00104 BC00104 V=100.0  +MOVJ EC00104
SREFP 3 C00105 BC00105  +REFP EC00105
CALL JOB:SEARCH-R1-S13D
SET P033 P006
SFTON3D P033
SMOVL C00106 BC00106 V=100.0  +MOVJ EC00106
SREFP 3 C00107 BC00107  +REFP EC00107
CALL JOB:SEARCH-R1-S13D
SET P033 P006
SFTON3D P033
SMOVL C00108 BC00108 V=100.0  +MOVJ EC00108
MOVL C00109 BC00109 V=400.0  +MOVJ EC00109 VJ=100.00
SFTOF3D
SMOVL C00110 BC00110 V=400.0  +MOVJ EC00110
SMOVL C00111 BC00111 V=166.7  +MOVJ EC00111
SMOVL C00112 BC00112 V=100.0  +MOVJ EC00112
SREFP 3 C00113 BC00113  +REFP EC00113
CALL JOB:SEARCH-R1-S13D
SET P034 P006
SFTON3D P034
SMOVL C00114 BC00114 V=100.0  +MOVJ EC00114
SMOVL C00115 BC00115 V=100.0  +MOVJ EC00115
SREFP 3 C00116 BC00116  +REFP EC00116
CALL JOB:SEARCH-R1-S13D
SET P034 P006
SFTON3D P034
SMOVL C00117 BC00117 V=100.0  +MOVJ EC00117
SFTOF3D
MOVL C00118 BC00118 V=1000.0  +MOVJ EC00118 VJ=100.00
MOVJ C00119 BC00119 VJ=100.00  +MOVJ EC00119 VJ=100.00
SMOVL C00120 BC00120 V=1000.0  +MOVJ EC00120
SMOVL C00121 BC00121 V=1000.0  +MOVJ EC00121
SMOVL C00122 BC00122 V=1000.0  +MOVJ EC00122
SMOVL C00123 BC00123 V=166.7  +MOVJ EC00123
SMOVL C00124 BC00124 V=100.0  +MOVJ EC00124
SREFP 3 C00125 BC00125  +REFP EC00125
CALL JOB:SEARCH-R1-S13D
SET P035 P006
SFTON3D P035
SMOVL C00126 BC00126 V=100.0  +MOVJ EC00126
SREFP 3 C00127 BC00127  +REFP EC00127
CALL JOB:SEARCH-R1-S13D
SET P035 P006
SFTON3D P035
SMOVL C00128 BC00128 V=100.0  +MOVJ EC00128
MOVL C00129 BC00129 V=400.0  +MOVJ EC00129 VJ=100.00
SFTOF3D
SMOVL C00130 BC00130 V=1000.0  +MOVJ EC00130
SMOVL C00131 BC00131 V=166.7  +MOVJ EC00131
SMOVL C00132 BC00132 V=100.0  +MOVJ EC00132
SREFP 3 C00133 BC00133  +REFP EC00133
CALL JOB:SEARCH-R1-S13D
SET P036 P006
SFTON3D P036
SMOVL C00134 BC00134 V=100.0  +MOVJ EC00134
SREFP 3 C00135 BC00135  +REFP EC00135
CALL JOB:SEARCH-R1-S13D
SET P036 P006
SFTON3D P036
SMOVL C00136 BC00136 V=100.0  +MOVJ EC00136
SFTOF3D
MOVL C00137 BC00137 V=400.0  +MOVJ EC00137 VJ=100.00
SMOVL C00138 BC00138 V=166.7  +MOVJ EC00138
SMOVL C00139 BC00139 V=100.0  +MOVJ EC00139
SREFP 3 C00140 BC00140  +REFP EC00140
CALL JOB:SEARCH-R1-S13D
SET P038 P006
SFTON3D P038
SMOVL C00141 BC00141 V=100.0  +MOVJ EC00141
SREFP 3 C00142 BC00142  +REFP EC00142
CALL JOB:SEARCH-R1-S13D
SET P038 P006
SFTON3D P038
SMOVL C00143 BC00143 V=100.0  +MOVJ EC00143
MOVL C00144 BC00144 V=400.0  +MOVJ EC00144 VJ=100.00
SFTOF3D
SMOVL C00145 BC00145 V=1000.0  +MOVJ EC00145
SMOVL C00146 BC00146 V=166.7  +MOVJ EC00146
SMOVL C00147 BC00147 V=100.0  +MOVJ EC00147
SREFP 3 C00148 BC00148  +REFP EC00148
CALL JOB:SEARCH-R1-S13D
SET P037 P006
SFTON3D P037
SMOVL C00149 BC00149 V=100.0  +MOVJ EC00149
SREFP 3 C00150 BC00150  +REFP EC00150
CALL JOB:SEARCH-R1-S13D
SET P037 P006
SFTON3D P037
SMOVL C00151 BC00151 V=100.0  +MOVJ EC00151
SREFP 3 C00152 BC00152  +REFP EC00152
CALL JOB:SEARCH-R1-S13D
SET P037 P006
SMOVL C00153 BC00153 V=100.0  +MOVJ EC00153
MOVL C00154 BC00154 V=400.0  +MOVJ EC00154 VJ=100.00
SMOVL C00155 BC00155 V=400.0  +MOVJ EC00155
MACRO1 MJ#(0) ARGF14
SFTON3D P037
SMOVL C00156 BC00156 V=100.0 PL=0  +MOVJ EC00156
ARCON
SMOVL C00157 BC00157 V=10.0  +MOVJ EC00157
SMOVL C00158 BC00158 V=10.0  +MOVJ EC00158
SMOVC C00159 BC00159 V=10.0  +MOVJ EC00159
SMOVC C00160 BC00160 V=10.0  +MOVJ EC00160
SMOVC C00161 BC00161 V=10.0  +MOVJ EC00161
SMOVL C00162 BC00162 V=10.0  +MOVJ EC00162
SMOVL C00163 BC00163 V=10.0  +MOVJ EC00163
ARCOF
SMOVL C00164 BC00164 V=166.7  +MOVJ EC00164
SFTOF3D
MOVJ C00165 BC00165 VJ=100.00  +MOVJ EC00165 VJ=100.00
MOVJ C00166 BC00166 VJ=100.00  +MOVJ EC00166 VJ=100.00
MOVJ C00167 BC00167 VJ=100.00  +MOVJ EC00167 VJ=100.00
MACRO1 MJ#(0) ARGF10
SFTON3D P035
SMOVL C00168 BC00168 V=166.7  +MOVJ EC00168
ARCON
SMOVL C00169 BC00169 V=6.7  +MOVJ EC00169
MOVL C00170 BC00170 V=6.7  +MOVJ EC00170 VJ=100.00
ARCOF
SMOVL C00171 BC00171 V=166.7  +MOVJ EC00171
SFTOF3D
SMOVL C00172 BC00172 V=166.7  +MOVJ EC00172
SFTON3D P036
SMOVL C00173 BC00173 V=166.7  +MOVJ EC00173
ARCON
SMOVL C00174 BC00174 V=5.8  +MOVJ EC00174
SMOVL C00175 BC00175 V=5.8  +MOVJ EC00175
ARCOF
SMOVL C00176 BC00176 V=166.7  +MOVJ EC00176
SFTOF3D
SMOVL C00177 BC00177 V=166.7  +MOVJ EC00177
SFTON3D P038
SMOVL C00178 BC00178 V=166.7  +MOVJ EC00178
ARCON
SMOVL C00179 BC00179 V=7.5  +MOVJ EC00179
ARCOF
SFTOF3D
MOVL C00180 BC00180 V=166.7  +MOVJ EC00180 VJ=80.00
MOVL C00181 BC00181 V=166.7  +MOVJ EC00181 VJ=80.00
SFTON3D P038
MOVL C00182 BC00182 V=166.7  +MOVJ EC00182 VJ=80.00
ARCON
MOVL C00183 BC00183 V=7.5  +MOVJ EC00183 VJ=80.00
ARCOF
MOVL C00184 BC00184 V=166.7  +MOVJ EC00184 VJ=80.00
SMOVL C00185 BC00185 V=166.7  +MOVJ EC00185
SFTOF3D
SMOVL C00186 BC00186 V=666.7  +MOVJ EC00186
SMOVL C00187 BC00187 V=666.7  +MOVJ EC00187
SMOVL C00188 BC00188 V=1000.0  +MOVJ EC00188
SMOVL C00189 BC00189 V=1000.0  +MOVJ EC00189
SMOVL C00190 BC00190 V=1000.0  +MOVJ EC00190
SMOVL C00191 BC00191 V=1000.0  +MOVJ EC00191
SFTON3D P033
SMOVL C00192 BC00192 V=250.0  +MOVJ EC00192
ARCON
SMOVL C00193 BC00193 V=5.8  +MOVJ EC00193
SMOVL C00194 BC00194 V=5.8  +MOVJ EC00194
ARCOF
SFTOF3D
SMOVL C00195 BC00195 V=166.7  +MOVJ EC00195
SMOVL C00196 BC00196 V=166.7  +MOVJ EC00196
SFTON3D P033
SMOVL C00197 BC00197 V=166.7  +MOVJ EC00197
ARCON
SMOVL C00198 BC00198 V=5.8  +MOVJ EC00198
SMOVL C00199 BC00199 V=5.8  +MOVJ EC00199
ARCOF
SMOVL C00200 BC00200 V=250.0  +MOVJ EC00200
MACRO1 MJ#(0) ARGF6
SMOVL C00201 BC00201 V=250.0  +MOVJ EC00201
ARCON
TIMER T=2.00
ARCOF
MOVJ C00202 BC00202 VJ=100.00  +MOVJ EC00202 VJ=100.00
MOVJ C00203 BC00203 VJ=100.00  +MOVJ EC00203 VJ=100.00
MACRO1 MJ#(0) ARGF9
SMOVL C00204 BC00204 V=250.0  +MOVJ EC00204
ARCON
SMOVL C00205 BC00205 V=7.5  +MOVJ EC00205
ARCOF
SMOVL C00206 BC00206 V=7.5  +MOVJ EC00206
ARCON
SMOVL C00207 BC00207 V=7.5  +MOVJ EC00207
ARCOF
SMOVL C00208 BC00208 V=250.0  +MOVJ EC00208
SMOVL C00209 BC00209 V=250.0  +MOVJ EC00209
SFTON3D P031
SMOVL C00210 BC00210 V=250.0  +MOVJ EC00210
ARCON
SMOVL C00211 BC00211 V=6.7  +MOVJ EC00211
ARCOF
SMOVL C00212 BC00212 V=133.3  +MOVJ EC00212
SMOVL C00213 BC00213 V=133.3  +MOVJ EC00213
ARCON
SMOVL C00214 BC00214 V=8.3  +MOVJ EC00214
SMOVL C00215 BC00215 V=8.3  +MOVJ EC00215
ARCOF
SMOVL C00216 BC00216 V=250.0  +MOVJ EC00216
MOVJ C00217 BC00217 VJ=100.00  +MOVJ EC00217 VJ=100.00
SFTOF3D
MOVJ C00218 BC00218 VJ=100.00  +MOVJ EC00218 VJ=100.00
MOVJ C00219 BC00219 VJ=100.00  +MOVJ EC00219 VJ=100.00
SFTON3D P032
SMOVL C00220 BC00220 V=250.0  +MOVJ EC00220
MACRO1 MJ#(0) ARGF14
ARCON
SMOVL C00221 BC00221 V=10.0  +MOVJ EC00221
SMOVC C00222 BC00222 V=10.0  +MOVJ EC00222
SMOVC C00223 BC00223 V=10.0  +MOVJ EC00223
SMOVC C00224 BC00224 V=10.0  +MOVJ EC00224
SMOVL C00225 BC00225 V=8.3  +MOVJ EC00225
ARCOF
SMOVL C00226 BC00226 V=250.0  +MOVJ EC00226
SFTOF3D
SMOVL C00227 BC00227 V=666.7  +MOVJ EC00227
MOVJ C00228 BC00228 VJ=100.00  +MOVJ EC00228 VJ=100.00
SFTON3D P021
SMOVL C00229 BC00229 V=250.0  +MOVJ EC00229
ARCON
SMOVL C00230 BC00230 V=10.0  +MOVJ EC00230
SMOVL C00231 BC00231 V=10.0  +MOVJ EC00231
ARCOF
SMOVL C00232 BC00232 V=250.0  +MOVJ EC00232
SFTOF3D
SMOVL C00233 BC00233 V=833.3  +MOVJ EC00233
SMOVL C00234 BC00234 V=833.3  +MOVJ EC00234
SMOVL C00235 BC00235 V=833.3  +MOVJ EC00235
SMOVL C00236 BC00236 V=833.3  +MOVJ EC00236
SFTON3D P027
SMOVL C00237 BC00237 V=250.0  +MOVJ EC00237
ARCON
SMOVL C00238 BC00238 V=10.0  +MOVJ EC00238
SMOVL C00239 BC00239 V=10.0  +MOVJ EC00239
SMOVL C00240 BC00240 V=10.0  +MOVJ EC00240
ARCOF
SMOVL C00241 BC00241 V=333.3  +MOVJ EC00241
SFTOF3D
SMOVL C00242 BC00242 V=333.3  +MOVJ EC00242
SMOVL C00243 BC00243 V=333.3  +MOVJ EC00243
SFTON3D P025
SMOVL C00244 BC00244 V=250.0  +MOVJ EC00244
ARCON
SFTON3D P024
SMOVL C00245 BC00245 V=10.0  +MOVJ EC00245
SMOVL C00246 BC00246 V=10.0  +MOVJ EC00246
ARCOF
SMOVL C00247 BC00247 V=250.0  +MOVJ EC00247
SMOVL C00248 BC00248 V=833.3  +MOVJ EC00248
SMOVL C00249 BC00249 V=833.3  +MOVJ EC00249
SMOVL C00250 BC00250 V=833.3  +MOVJ EC00250
SMOVL C00251 BC00251 V=333.3  +MOVJ EC00251
SFTON3D P022
SMOVL C00252 BC00252 V=166.7  +MOVJ EC00252
ARCON
SMOVL C00253 BC00253 V=10.0  +MOVJ EC00253
SMOVL C00254 BC00254 V=10.0  +MOVJ EC00254
SFTON3D P023
SMOVL C00255 BC00255 V=10.0  +MOVJ EC00255
SMOVL C00256 BC00256 V=10.0  +MOVJ EC00256
ARCOF
SMOVL C00257 BC00257 V=250.0  +MOVJ EC00257
SFTOF3D
MOVJ C00258 BC00258 VJ=100.00  +MOVJ EC00258 VJ=100.00
MOVJ C00259 BC00259 VJ=100.00  +MOVJ EC00259 VJ=100.00
MOVJ C00260 BC00260 VJ=100.00  +MOVJ EC00260 VJ=100.00
MOVJ C00261 BC00261 VJ=100.00  +MOVJ EC00261 VJ=100.00
SFTON3D P025
SMOVL C00262 BC00262 V=250.0  +MOVJ EC00262
ARCON
SFTON3D P026
SMOVL C00263 BC00263 V=10.0  +MOVJ EC00263
ARCOF
SMOVL C00264 BC00264 V=400.0  +MOVJ EC00264
SFTOF3D
MOVJ C00265 BC00265 VJ=100.00  +MOVJ EC00265 VJ=100.00
MOVJ C00266 BC00266 VJ=100.00  +MOVJ EC00266 VJ=100.00
MOVJ C00267 BC00267 VJ=100.00  +MOVJ EC00267 VJ=100.00
SFTON3D P021
SMOVL C00268 BC00268 V=400.0  +MOVJ EC00268
ARCON
SFTON3D P022
SMOVL C00269 BC00269 V=10.0  +MOVJ EC00269
ARCOF
SFTOF3D
SMOVL C00270 BC00270 V=250.0  +MOVJ EC00270
SMOVL C00271 BC00271 V=833.3  +MOVJ EC00271
SMOVL C00272 BC00272 V=833.3  +MOVJ EC00272
END
